FUNCTION_BLOCK UA_ConnectWrapper IMPLEMENTS I_OPCUA_Connect
VAR_INPUT
END_VAR
VAR_OUTPUT
END_VAR
VAR
	uaConnect : UA_Connect;
END_VAR

{warning 'add method implementation '}
METHOD start : BOOL
VAR_INPUT
	Execute					: BOOL;
	ServerUrl				: STRING(MAX_STRING_LENGTH);
	SessionConnectInfo		: Tc3_PLCopen_OpcUa.ST_UASessionConnectInfo;
	Timeout					: TIME := DEFAULT_ADS_TIMEOUT;
END_VAR
VAR_OUTPUT
	ConnectionHdl			: DWORD;
	Done					: BOOL;
	Busy					: BOOL;
	Error					: BOOL;
	ErrorID					: DWORD;
END_VAR
uaConnect(Execute					:= Execute,
          ServerUrl				:= ServerUrl	,
          SessionConnectInfo		:= SessionConnectInfo,
          Timeout					:= Timeout,
		  ConnectionHdl			=> ConnectionHdl,
		  Done					=> Done,
          Busy					=> Busy,
          Error					=> Error,
          ErrorID				=> ErrorID
		  );
END_METHOD

END_FUNCTION_BLOCK

(* stored: Version 1.1.0.1, ProductVersion 3.1.4024.9
   POU UA_ConnectWrapper: Id {99419b85-d4bf-4b2c-bdc6-398c4daf6560}, SpecialFunc None
   Method start: Id {14decb79-d22a-4785-bd37-bad7aca342af} *)
